{attribute 'call_after_init'}
FUNCTION_BLOCK fb_CalCulateAccumulation_Test EXTENDS TcUnit.FB_TestSuite IMPLEMENTS TcUnit.I_TestResults

VAR
	fbCalEnergy : FB_CalCulateAccumulation;
	CurrentTime : TIMESTRUCT;

END_VAR

fbCalEnergy( lrAccumulator := pmDev.DB06_02_5500.Basic.RealEnergy_IntoLoad,
				CurrentTime := CurrentTime) ;// lv04

METHOD FB_init : BOOL
VAR_INPUT
    bInitRetains : BOOL; // if TRUE, the retain variables are initialized (warm start / cold start)
    bInCopyCode : BOOL;  // if TRUE, the instance afterwards gets moved into the copy code (online change)
END_VAR
END_METHOD

END_FUNCTION_BLOCK

(* stored: Version 1.1.0.1, ProductVersion 3.1.4024.12
   POU fb_CalCulateAccumulation_Test: Id {1efb4bea-9641-4821-84f7-351ca5d4cc7a}, SpecialFunc None
   Method FB_init: Id {47b08a03-9ccf-4c17-8eab-477843e639b4} *)
